// TIA Portal project "template_V21" (V21)
// template for the blocks

(* hardware
DEVICE "S7-1200 station_1"  S7-1200 Station
   slot 0: "Rack_0"  S7-1200 Rack  Rack  V1.0
   slot 1: "PLC_1"  CPU 1214C DC/DC/DC  6ES7 214-1AG40-0XB0  V4.2
DEVICE "HMI_1"  TP700 Comfort
   slot 0: "HMI_1"  TP700 Comfort  6AV2 124-0GC01-0AX0  17.0.0.0
   slot 1: "HMI_RT_1"  TP700 Comfort  6AV2 124-0GC01-0AX0  17.0.0.0
   slot 5: "HMI_1.IE_CP_1"  PROFINET Interface  17.0.0.0
      slot 1: "PROFINET Interface_1"  PROFINET Interface
         slot 1: "Port_1"  Port
         slot 2: "Port_2"  Port
   slot 7: "HMI_1.MPI/DP_CP_1"  MPI/DP Interface  17.0.0.0
*)

// ===== PLC "PLC_1"  CPU 1214C DC/DC/DC =====

ORGANIZATION_BLOCK "system.Main"   // OB1, SCL, ProgramCycle
TITLE = "Main Program Sweep (Cycle)"
{ S7_Optimized_Access := 'TRUE' }
VERSION : 0.1
   VAR_INPUT
      Initial_Call : Bool;   // Initial call of this OB
      Remanence : Bool;   // =True, if remanent data are available
   END_VAR
BEGIN
   "Main"();
END_ORGANIZATION_BLOCK

ORGANIZATION_BLOCK "system.Startup"   // OB100, SCL, Startup
TITLE = "Complete Restart"
{ S7_Optimized_Access := 'TRUE' }
VERSION : 0.1
   VAR_INPUT
      LostRetentive : Bool;   // True if retentive data are lost
      LostRTC : Bool;   // True if date and time are lost
   END_VAR
BEGIN
   "Startup"(#LostRetentive=#LostRetentive, #LostRTC=#LostRTC);
END_ORGANIZATION_BLOCK

(* ===== HMI "HMI_RT_1" =====
system functions are stored by id; their names below are inferred from use
connection "HMI_Connection_1": ETHERNET, S7_1200_OMS

screen "Root screen" 800x480, template "Template_1"
   TextField "HmiScreenItemData_3" at 80,225 size 640x25; Text 'Welcome to HMI_1 (TP700 Comfort)!'
   Button "HmiScreenItemData" at 36,36 size 159x47; TextOff 'manual'; PictureOff "Navigates to manual for TP700 Comfort 17.0.0.0"; PictureOn "Navigates to manual for TP700 Comfort 17.0.0.0"
      on Release: ActivateScreen("manual", 0)
   Button "HmiScreenItemData_1" at 36,95 size 159x47; TextOff 'auto'; PictureOff "Navigates to auto for TP700 Comfort 17.0.0.0"; PictureOn "Navigates to auto for TP700 Comfort 17.0.0.0"
      on Release: ActivateScreen("auto", 0)
   Button "HmiScreenItemData_2" at 36,154 size 159x47; TextOff 'override'; PictureOff "Navigates to override for TP700 Comfort 17.0.0.0"; PictureOn "Navigates to override for TP700 Comfort 17.0.0.0"
      on Release: ActivateScreen("override", 0)

screen "manual" 800x480, template "Template_1"
   TextField "HmiScreenItemData" at 80,225 size 640x25; Text 'manual'
   Button "Back" at 1,1 size 159x47; TextOff 'Back'
      on Release: ActivateScreen("Root screen", 0)

screen "auto" 800x480, template "Template_1"
   TextField "HmiScreenItemData" at 80,225 size 640x25; Text 'auto'
   Button "Back" at 1,1 size 159x47; TextOff 'Back'
      on Release: ActivateScreen("Root screen", 0)
   Button "HmiScreenItemData_1" at 36,95 size 159x47; TextOff 'autohome'; PictureOff "Navigates to autohome for TP700 Comfort 17.0.0.0"; PictureOn "Navigates to autohome for TP700 Comfort 17.0.0.0"
      on Release: ActivateScreen("autohome", 0)
   Button "HmiScreenItemData_2" at 36,154 size 159x47; TextOff 'normal operation'; PictureOff "Navigates to normal operation for TP700 Comfort 17.0.0.0"; PictureOn "Navigates to normal operation for TP700 Comfort 17.0.0.0"
      on Release: ActivateScreen("normal operation", 0)

screen "autohome" 800x480, template "Template_1"
   TextField "HmiScreenItemData" at 80,225 size 640x25; Text 'autohome'
   Button "Back" at 1,1 size 159x47; TextOff 'Back'
      on Release: ActivateScreen("auto", 0)

screen "normal operation" 800x480, template "Template_1"
   TextField "HmiScreenItemData" at 80,225 size 640x25; Text 'normal operation'
   Button "Back" at 1,1 size 159x47; TextOff 'Back'
      on Release: ActivateScreen("auto", 0)

screen "override" 800x480, template "Template_1"
   TextField "HmiScreenItemData" at 80,225 size 640x25; Text 'override'
   Button "Back" at 1,1 size 159x47; TextOff 'Back'
      on Release: ActivateScreen("Root screen", 0)
*)